TYPE ST_St040_IO_IN :
STRUCT
END_STRUCT
END_TYPE

(* stored: Version 1.1.0.1
   DUT ST_St040_IO_IN: Id {74728f09-4a98-4122-8d4e-1e63a12abb25} *)
